{attribute 'qualified_only'}
VAR_GLOBAL CONSTANT
	
	(*Checks whether the TC3 event logger is set as standard in the XTS prosessing unit.*)
	B_MSG_IF_TC3EVENTLOGGER_IS_NOT_DEFAULT: BOOL := TRUE;	

	MAX_MOVER_PER_SYSTEM : UINT := 50;
	MAX_MOTORS_PER_SYSTEM : UINT := 100;
	STATISTIC_AVG_PERIOD : TIME := T#10S;
END_VAR

(* stored: Version 1.1.0.1, ProductVersion 3.1.4024.12
   GVL XtsParameterlist: Id {a0a7e988-ac8b-4d02-827c-c315d3a6afd8}, ParameterList True *)
